ABB RAPID module: Wobj_base_nest_legs.mod

MODULE Wobj_base_nest_legs
	! Points are read in order of declaration.
  ! Please do not change the order of points!

  LOCAL PERS robtarget pWobj_U_PointX1:=[[1366.667,-46.64455,-444.0839],[0.000427774182753637,-0.738901317119598,-0.673747301101685,-0.0094472412019968],[-1,0,1,0],[9E+09,9E+09,9E+09,9E+09,9E+09,9E+09]];
	LOCAL PERS robtarget pWobj_U_PointX2:=[[682.7925,-628.1551,-458.5991],[0.000454275461379439,-0.738939583301544,-0.673705220222473,-0.00945208501070738],[-1,0,0,0],[9E+09,9E+09,9E+09,9E+09,9E+09,9E+09]];
	LOCAL PERS robtarget pWobj_U_PointY1:=[[1893.753,-664.0765,-452.493],[0.000433340610470623,-0.738940000534058,-0.673704743385315,-0.00945510528981686],[-1,0,0,0],[9E+09,9E+09,9E+09,9E+09,9E+09,9E+09]];

ENDMODULE
